{attribute 'linkalways'} 
{attribute 'no_explicit_call' := 'This FB is a CLASS and must be accessed using methods or properties'}
{attribute 'enable_dynamic_creation'}
FUNCTION_BLOCK NodeExecuteBeginEvent EXTENDS Disposable IMPLEMENTS I_NodeExecuteBeginEvent
VAR
	_target : I_Node;
	_cpuCounterLowBytes : UDINT;
	_cpuCounterHighBytes : UDINT;
END_VAR

PROPERTY PUBLIC CpuCounterHighBytes : UDINT
GET
CpuCounterHighBytes := _cpuCounterHighBytes;
END_GET
END_PROPERTY

PROPERTY PUBLIC CpuCounterLowBytes : UDINT
GET
CpuCounterLowBytes := _cpuCounterLowBytes;
END_GET
END_PROPERTY

METHOD FB_init : BOOL
VAR_INPUT
	bInitRetains : BOOL; // if TRUE, the retain variables are initialized (warm start / cold start)
	bInCopyCode : BOOL;  // if TRUE, the instance afterwards gets moved into the copy code (online change)
	Target : I_Node;
END_VAR
VAR
	getCount : GETCPUCOUNTER;
END_VAR
_target := Target;
getCount(cpuCntLoDW => _cpuCounterLowBytes, cpuCntHiDW => _cpuCounterHighBytes);
END_METHOD

PROPERTY PUBLIC Target : I_Node
GET
Target := _target;
END_GET
END_PROPERTY

END_FUNCTION_BLOCK

(* stored: Version 1.1.0.1, ProductVersion 3.1.4024.12
   POU NodeExecuteBeginEvent: Id {099dccbd-4b03-47d2-99bd-82fca18aee68}, SpecialFunc None
   Folder Constructor: Id {1a6c8cd5-bcb5-4c10-b56d-6c473d81d706}
   Property CpuCounterHighBytes: Id {cedc6650-b823-42b9-aa58-ff8fb90d7bb7}
   Get Get: Id {a8c57d2d-cb61-4738-b92e-97af1cc14593}
   Property CpuCounterLowBytes: Id {57f83f18-ddd0-4b38-aac8-92c36132de94}
   Get Get: Id {ed4bec57-ac38-4207-86c4-c621876ab65a}
   Method FB_init: Id {4ec819db-f346-4b43-8801-a31bd8c2496d}
   Property Target: Id {ed5dfaf5-a388-4a64-96b4-f9ac8b1cd611}
   Get Get: Id {a32eee2b-f93d-45f0-a7a8-fda0a40cdb68} *)
